{attribute 'linkalways'} 
{attribute 'no_explicit_call' := 'This FB is a CLASS and must be accessed using methods or properties'}
{attribute 'enable_dynamic_creation'}
FUNCTION_BLOCK _ETcVnKeypointDetectionTypeFAST EXTENDS EnumDatatypeBase
VAR
	localData : ETcVnKeypointDetectionTypeFAST;
	activeData : REFERENCE TO ETcVnKeypointDetectionTypeFAST;
	enumBaseDatatype : _DINT(localData);
END_VAR

METHOD PRIVATE AddLocalEnumeration
VAR_INPUT
	Enumeration : T_MAXSTRING;
	Value : ETcVnKeypointDetectionTypeFAST;
END_VAR
AddEnumeration(Enumeration, Value);
END_METHOD

PROPERTY PUBLIC Address : PVOID
GET
Address := ADR(activeData);
END_GET
END_PROPERTY

METHOD PUBLIC ClearReference
VAR_INPUT
END_VAR
activeData REF= localData;
SetBaseDatatypeReference();
END_METHOD

METHOD PUBLIC Clone : I_Datatype
VAR
    pClone : POINTER TO _ETcVnKeypointDetectionTypeFAST;
END_VAR
pClone := __NEW(_ETcVnKeypointDetectionTypeFAST(InitialValue := Value));
Clone := pClone^;
END_METHOD

METHOD FB_init : BOOL
VAR_INPUT
	bInitRetains : BOOL; // if TRUE, the retain variables are initialized (warm start / cold start)
	bInCopyCode : BOOL;  // if TRUE, the instance afterwards gets moved into the copy code (online change)
	InitialValue : ETcVnKeypointDetectionTypeFAST;
END_VAR
localData := InitialValue;
AddBaseDatatype(enumBaseDatatype);
ClearReference();

AddLocalEnumeration('TCVN_KDT_FAST_5_8', ETcVnKeypointDetectionTypeFAST.TCVN_KDT_FAST_5_8);
AddLocalEnumeration('TCVN_KDT_FAST_7_12', ETcVnKeypointDetectionTypeFAST.TCVN_KDT_FAST_7_12);
AddLocalEnumeration('TCVN_KDT_FAST_9_16', ETcVnKeypointDetectionTypeFAST.TCVN_KDT_FAST_9_16);
END_METHOD

PROPERTY PUBLIC Identifier : T_MAXSTRING
GET
Identifier := 'ETcVnKeypointDetectionTypeFAST';
END_GET
END_PROPERTY

METHOD IsEnumeratorValueEqual : BOOL
VAR_INPUT
	Enumerator : I_KeyValueForwardEnumerator;
END_VAR
VAR
	storedValue : ETcVnKeypointDetectionTypeFAST;
END_VAR
IF NOT Enumerator.TryGet(storedValue) THEN
	RETURN;
END_IF

IsEnumeratorValueEqual := storedValue = activeData;
END_METHOD

METHOD PUBLIC MakeReferenceTo
VAR_INPUT
	ReferenceTarget : REFERENCE TO ETcVnKeypointDetectionTypeFAST;
END_VAR
activeData REF= ReferenceTarget;
SetBaseDatatypeReference();
END_METHOD

METHOD PROTECTED SetBaseDatatypeReference
VAR_INPUT
END_VAR
enumBaseDatatype.MakeReferenceTo(activeData);
END_METHOD

PROPERTY PUBLIC Size : UDINT
GET
Size := SIZEOF(activeData);
END_GET
END_PROPERTY

METHOD TryMakeReferenceTo : BOOL
VAR_INPUT
	Target : I_Datatype;
END_VAR
VAR
	targetAsEnum : I_EnumDatatype;
	pTargetData : POINTER TO ETcVnKeypointDetectionTypeFAST;
END_VAR
IF NOT Target.TryResolveAsEnumDatatype(targetAsEnum) THEN
	RETURN;
END_IF

IF targetAsEnum.Identifier <> Identifier THEN
	RETURN;
END_IF

pTargetData := Target.Address;
activeData REF= pTargetData^;
SetBaseDatatypeReference();
TryMakeReferenceTo := TRUE;
END_METHOD

PROPERTY PUBLIC Value : ETcVnKeypointDetectionTypeFAST
GET
Value := activeData;
END_GET
SET
activeData := Value;
END_SET
END_PROPERTY

END_FUNCTION_BLOCK

(* stored: Version 1.1.0.1
   POU _ETcVnKeypointDetectionTypeFAST: Id {26b6417e-5de4-44eb-8b13-1a38f4ffa521}, SpecialFunc None
   Folder Constructor: Id {922d1360-4f67-45a7-9bc3-c593a67d166d}
   Folder Private: Id {ad6ab5ef-0e97-45ab-8972-b9a8b9ff5be4}
   Folder Protected: Id {740bd1c7-16b6-45e6-8eb8-ef6e67cdf6d7}
   Method AddLocalEnumeration: Id {01eb5e13-69d4-4d9a-af16-29738f967490}
   Property Address: Id {0175d073-37a9-4e37-9721-6649f32fa2da}
   Get Get: Id {4059c712-e014-465e-beaf-362e6631fb65}
   Method ClearReference: Id {a39d0810-36dc-418d-818d-c8427a07f142}
   Method Clone: Id {6f076e83-d5b5-445b-9ba9-89193dd421d1}
   Method FB_init: Id {a42b32ae-9301-4a8a-adfb-bc43cebd3e0c}
   Property Identifier: Id {6f9d9c3e-3fb0-419d-8ff9-d6a5484241bd}
   Get Get: Id {8c81b2cb-70b6-4312-88e8-e19e78eb45f9}
   Method IsEnumeratorValueEqual: Id {69173549-1f04-453a-bdef-8010315fc109}
   Method MakeReferenceTo: Id {8f36b06f-0ad4-4d6a-88aa-c6cb6f0297dd}
   Method SetBaseDatatypeReference: Id {ab777e47-b2f3-4f38-b588-1c45ce54cb85}
   Property Size: Id {f8e637da-4a27-43c0-b63a-aa96e93e8608}
   Get Get: Id {692a1b1b-0b59-4f4b-800a-0031be9d3ee1}
   Method TryMakeReferenceTo: Id {19f27351-6789-44ea-99f2-1b92952fc5e0}
   Property Value: Id {3d6069ab-e822-403e-a18b-9e0aa802f9c1}
   Get Get: Id {15c798e0-ed3a-4bf0-a820-d50057eb673b}
   Set Set: Id {1d4e6508-664b-4ee0-908e-d029b693ca7e} *)
